Fanuc KAREL source: kc00036.KL

-- PROVISIONAL review KL for V1013-1; original PC SHA256 015f6f73968fc5cc2539566d75a1036071e2b3aae265819f65f0df982e3c7d9e
-- Incomplete behavior may be omitted. Consult companion uncertainty JSON. Do not deploy.
PROGRAM KC00036
%NOLOCKGROUP
BEGIN
  -- UNRESOLVED_PC offsets 5-15; opcodes 27,31,23
  -- UNRESOLVED_PC offsets 20-24; opcodes 7F
END KC00036
